// TIA Portal V19 export
FUNCTION "TOD_Pièces_List" : Void   // FC2, STL
BEGIN

NETWORK
TITLE = 
// BONNES PIECES DECALAGE

      OPN   "DB Bonnes Pièces";

//Pointeurs de 2 mémoires qui se suivent
      L     P#58.0;
      T     "Pointeur 1";
      L     P#60.0;
      T     "Pointeur 2";

//Compteur à 30 itérations
      L     30;
bcl1: T     "Compteur Bonnes Pièces";

//transfert JX à JX-1
      L     DBW ["Pointeur 1"];
      T     DBW ["Pointeur 2"];

//On retire 2 car double octet aux pointeurs pour avancer d'un jour
      L     "Pointeur 1";
      L     P#2.0;
      -D;
      T     "Pointeur 1";

      L     "Pointeur 2";
      L     P#2.0;
      -D;
      T     "Pointeur 2";

//Fin de la loop on charge le compteur et le loop enlève 1. Out si =0
      L     "Compteur Bonnes Pièces";
      LOOP  bcl1;


//Ajouter la variable avec Nb pièce de la journée
      L     "A CHANGER";
      T     "DB Bonnes Pièces"."Nb_J-1";

//Nouvelle Journée
      L     0;
      T     "A CHANGER";


NETWORK
TITLE = 
// PIECES NOIRES DECALAGE

      OPN   "DB Mauvaises Pièces";

//Pointeurs de 2 mémoires qui se suivent
      L     P#58.0;
      T     "Pointeur 1";
      L     P#60.0;
      T     "Pointeur 2";

//Compteur à 30 itérations
      L     30;
bcl2: T     "Compteur Mauvaises Pièces";

//transfert JX à JX-1
      L     DBW ["Pointeur 1"];
      T     DBW ["Pointeur 2"];

//On retire 2 car double octet aux pointeurs pour avancer d'un jour
      L     "Pointeur 1";
      L     P#2.0;
      -D;
      T     "Pointeur 1";

      L     "Pointeur 2";
      L     P#2.0;
      -D;
      T     "Pointeur 2";

//Fin de la loop on charge le compteur et le loop enlève 1. Out si =0
      L     "Compteur Mauvaises Pièces";
      LOOP  bcl2;


//Ajouter la variable avec Nb pièce de la journée
      L     "A CHANGER";
      T     "DB Mauvaises Pièces"."Nb_J-1";

//Nouvelle Journée
      L     0;
      T     "A CHANGER";

END_FUNCTION
